(* IEC 61131-3 sources: com.logicals.lc3.webinar/usRTS_RPMControl_iSOC/src_FB_LIB_SAFE/Bitstring/WORD, 10 files *)

(* ---- wAND_WORD_2.iecst ---- *)
NAMESPACE logicals.web.standard
NAMESPACE bitstring

/*
 * Function block wrapper for IEC 61131-3 AND<br>
 * IN1 =  1st value (WORD)<br>
 * IN2 =  2nd value (WORD)<br>
 * OUT = IN1 AND IN2 (WORD)<br>
 */
FUNCTION_BLOCK wAND_WORD_2
	{ vNameAlignment:="center"; altName:="&"; bgColor:="DodgerBlue"; width:=40; hideIONames; }
	VAR_INPUT
		IN1 : WORD;
		IN2 : WORD;
	END_VAR
	VAR_OUTPUT
		OUT: WORD;
	END_VAR

	OUT := AND(IN1:=IN1, IN2:=IN2, ENO=>ENO);
END_FUNCTION_BLOCK

END_NAMESPACE
END_NAMESPACE

(* ---- wAND_WORD_3.iecst ---- *)
NAMESPACE logicals.web.standard
NAMESPACE bitstring

/*
 * Function block wrapper for IEC 61131-3 AND<br>
 * IN1 =  1st value (WORD)<br>
 * IN2 =  2nd value (WORD)<br>
 * IN3 =  3rd value (WORD)<br>
 * OUT = IN1 AND IN2 AND IN3 (WORD)<br>
 */
FUNCTION_BLOCK wAND_WORD_3
	{ vNameAlignment:="center"; altName:="&"; bgColor:="DodgerBlue"; width:=40; hideIONames; }
	VAR_INPUT
		IN1 : WORD;
		IN2 : WORD;
		IN3 : WORD;
	END_VAR
	VAR_OUTPUT
		OUT: WORD;
	END_VAR

	OUT := AND(IN1:=IN1, IN2:=IN2, IN3:=IN3, ENO=>ENO);
END_FUNCTION_BLOCK

END_NAMESPACE
END_NAMESPACE

(* ---- wAND_WORD_4.iecst ---- *)
NAMESPACE logicals.web.standard
NAMESPACE bitstring

/*
 * Function block wrapper for IEC 61131-3 AND<br>
 * IN1 =  1st value (WORD)<br>
 * IN2 =  2nd value (WORD)<br>
 * IN3 =  3rd value (WORD)<br>
 * IN4 =  4th value (WORD)<br>
 * OUT = IN1 AND IN2 AND IN3 AND IN4 (WORD)<br>
 */
FUNCTION_BLOCK wAND_WORD_4
	{ vNameAlignment:="center"; altName:="&"; bgColor:="DodgerBlue"; width:=40; hideIONames; }
	VAR_INPUT
		IN1 : WORD;
		IN2 : WORD;
		IN3 : WORD;
		IN4 : WORD;
	END_VAR
	VAR_OUTPUT
		OUT: WORD;
	END_VAR

	OUT := AND(IN1:=IN1, IN2:=IN2, IN3:=IN3, IN4:=IN4, ENO=>ENO);
END_FUNCTION_BLOCK

END_NAMESPACE
END_NAMESPACE

(* ---- wNOT_WORD.iecst ---- *)
NAMESPACE logicals.web.standard
NAMESPACE bitstring

/*
 * Function block wrapper for IEC 61131-3 NOT<br>
 * IN = input (WORD)<br>
 * OUT = !IN (WORD)<br>
 */
FUNCTION_BLOCK wNOT_WORD
	{ vNameAlignment:="center"; altName:="NOT"; bgColor:="DodgerBlue"; width:=60; hideIONames; }
	VAR_INPUT
		IN : WORD;
	END_VAR
	VAR_OUTPUT
		OUT: WORD;
	END_VAR

	OUT := NOT(IN:=IN, ENO=>ENO);
END_FUNCTION_BLOCK

END_NAMESPACE
END_NAMESPACE

(* ---- wOR_WORD_2.iecst ---- *)
NAMESPACE logicals.web.standard
NAMESPACE bitstring

/*
 * Function block wrapper for IEC 61131-3 OR<br>
 * IN1 =  1st value (WORD)<br>
 * IN2 =  2nd value (WORD)<br>
 * OUT = IN1 OR IN2 (WORD)<br>
 */
FUNCTION_BLOCK wOR_WORD_2
	{ vNameAlignment:="center"; altName:=">=1"; bgColor:="DodgerBlue"; width:=40; hideIONames; }
	VAR_INPUT
		IN1 : WORD;
		IN2 : WORD;
	END_VAR
	VAR_OUTPUT
		OUT: WORD;
	END_VAR

	OUT := OR(IN1:=IN1, IN2:=IN2, ENO=>ENO);
END_FUNCTION_BLOCK

END_NAMESPACE
END_NAMESPACE

(* ---- wOR_WORD_3.iecst ---- *)
NAMESPACE logicals.web.standard
NAMESPACE bitstring

/*
 * Function block wrapper for IEC 61131-3 OR<br>
 * IN1 =  1st value (WORD)<br>
 * IN2 =  2nd value (WORD)<br>
 * IN3 =  3rd value (WORD)<br>
 * OUT = IN1 OR IN2 OR IN3 (WORD)<br>
 */
FUNCTION_BLOCK wOR_WORD_3
	{ vNameAlignment:="center"; altName:=">=1"; bgColor:="DodgerBlue"; width:=40; hideIONames; }
	VAR_INPUT
		IN1 : WORD;
		IN2 : WORD;
		IN3 : WORD;
	END_VAR
	VAR_OUTPUT
		OUT: WORD;
	END_VAR

	OUT := OR(IN1:=IN1, IN2:=IN2, IN3:=IN3, ENO=>ENO);
END_FUNCTION_BLOCK

END_NAMESPACE
END_NAMESPACE

(* ---- wOR_WORD_4.iecst ---- *)
NAMESPACE logicals.web.standard
NAMESPACE bitstring

/*
 * Function block wrapper for IEC 61131-3 OR<br>
 * IN1 =  1st value (WORD)<br>
 * IN2 =  2nd value (WORD)<br>
 * IN3 =  3rd value (WORD)<br>
 * IN4 =  4th value (WORD)<br>
 * OUT = IN1 OR IN2 OR IN3 OR IN4 (WORD)<br>
 */
FUNCTION_BLOCK wOR_WORD_4
	{ vNameAlignment:="center"; altName:=">=1"; bgColor:="DodgerBlue"; width:=40; hideIONames; }
	VAR_INPUT
		IN1 : WORD;
		IN2 : WORD;
		IN3 : WORD;
		IN4 : WORD;
	END_VAR
	VAR_OUTPUT
		OUT: WORD;
	END_VAR

	OUT := OR(IN1:=IN1, IN2:=IN2, IN3:=IN3, IN4:=IN4, ENO=>ENO);
END_FUNCTION_BLOCK

END_NAMESPACE
END_NAMESPACE

(* ---- wXOR_WORD_2.iecst ---- *)
NAMESPACE logicals.web.standard
NAMESPACE bitstring

/*
 * Function block wrapper for IEC 61131-3 XOR<br>
 * IN1 =  1st value (WORD)<br>
 * IN2 =  2nd value (WORD)<br>
 * OUT = IN1 XOR IN2 (WORD)<br>
 */
FUNCTION_BLOCK wXOR_WORD_2
	{ vNameAlignment:="center"; altName:="=2k+1"; bgColor:="DodgerBlue"; width:=50; hideIONames; }
	VAR_INPUT
		IN1 : WORD;
		IN2 : WORD;
	END_VAR
	VAR_OUTPUT
		OUT: WORD;
	END_VAR

	OUT := XOR(IN1:=IN1, IN2:=IN2, ENO=>ENO);
END_FUNCTION_BLOCK

END_NAMESPACE
END_NAMESPACE

(* ---- wXOR_WORD_3.iecst ---- *)
NAMESPACE logicals.web.standard
NAMESPACE bitstring

/*
 * Function block wrapper for IEC 61131-3 XOR<br>
 * IN1 =  1st value (WORD)<br>
 * IN2 =  2nd value (WORD)<br>
 * IN3 =  3rd value (WORD)<br>
 * OUT = IN1 XOR IN2 XOR IN3 (WORD)<br>
 */
FUNCTION_BLOCK wXOR_WORD_3
	{ vNameAlignment:="center"; altName:="=2k+1"; bgColor:="DodgerBlue"; width:=50; hideIONames; }
	VAR_INPUT
		IN1 : WORD;
		IN2 : WORD;
		IN3 : WORD;
	END_VAR
	VAR_OUTPUT
		OUT: WORD;
	END_VAR

	OUT := XOR(IN1:=IN1, IN2:=IN2, IN3:=IN3, ENO=>ENO);
END_FUNCTION_BLOCK

END_NAMESPACE
END_NAMESPACE

(* ---- wXOR_WORD_4.iecst ---- *)
NAMESPACE logicals.web.standard
NAMESPACE bitstring

/*
 * Function block wrapper for IEC 61131-3 XOR<br>
 * IN1 =  1st value (WORD)<br>
 * IN2 =  2nd value (WORD)<br>
 * IN3 =  3rd value (WORD)<br>
 * IN4 =  4th value (WORD)<br>
 * OUT = IN1 XOR IN2 XOR IN3 XOR IN4 (WORD)<br>
 */
FUNCTION_BLOCK wXOR_WORD_4
	{ vNameAlignment:="center"; altName:="=2k+1"; bgColor:="DodgerBlue"; width:=50; hideIONames; }
	VAR_INPUT
		IN1 : WORD;
		IN2 : WORD;
		IN3 : WORD;
		IN4 : WORD;
	END_VAR
	VAR_OUTPUT
		OUT: WORD;
	END_VAR

	OUT := XOR(IN1:=IN1, IN2:=IN2, IN3:=IN3, IN4:=IN4, ENO=>ENO);
END_FUNCTION_BLOCK

END_NAMESPACE
END_NAMESPACE
